PROGRAM FBD_Controls_Overview
VAR
	fbBlock_1: FB_BlockPad;
	fbBlock_2: FB_BlockPad;
END_VAR

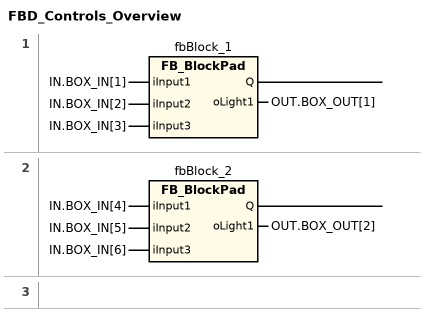
// NETWORK 1
fbBlock_1(
    iInput1 := IN.BOX_IN[1],
    iInput2 := IN.BOX_IN[2],
    iInput3 := IN.BOX_IN[3],
    oLight1 => OUT.BOX_OUT[1]); // FB_BlockPad

// NETWORK 2
fbBlock_2(
    iInput1 := IN.BOX_IN[4],
    iInput2 := IN.BOX_IN[5],
    iInput3 := IN.BOX_IN[6],
    oLight1 => OUT.BOX_OUT[2]); // FB_BlockPad

// NETWORK 3

END_PROGRAM

(* stored: Version 1.1.0.1, ProductVersion 3.1.4024.10
   POU FBD_Controls_Overview: Id {5015793d-548e-4713-ad62-be76714ca000}, SpecialFunc None *)
